{attribute 'GeneratedUsingTerminal: EK1122-0000-0018'}
{attribute addProperty BoxType "EK1122-0000-0018"}
{attribute addProperty Id "Beckhoff_EP9xxxsub_EK1100EK1100_1FC0878B2A_0001_EP9128_0020_0016A_0001_EP9128_0020_0016_C3F65AAB537"}
{attribute addProperty CRC "1150195516"}
{attribute addProperty Size "539"}
TYPE Beckhoff_EP9xxxEK1122_448E973C EXTENDS EK1122_1FC0878B :
STRUCT
	{attribute addProperty Name "Beckhoff_EP9xxxsub_EK1100"}
	{attribute addProperty PreviousPort "Beckhoff EP9xxxEK1122 : D"}
	Beckhoff_EP9xxxsub_EK1100 : EK1100_1FC0878B;
	{attribute addProperty Name "A_0001_EP9128_0020_0016"}
	{attribute addProperty PreviousPort "Beckhoff EP9xxxsub EK1100 : C"}
	A_0001_EP9128_0020_0016 : A_0001_EP9128_0020_0016_C3F65AAB;
END_STRUCT
END_TYPE

(* stored: Version 1.2.0.0, ProductVersion 3.1.4024.9
   DUT Beckhoff_EP9xxxEK1122_448E973C: Id {102e9550-a3bd-4f86-a25a-105051951f9f} *)
